// TIA Portal V17 export
// export: Created 2025-06-26T07:49:50.4539602Z, ExportSetting WithDefaults, DisplayName Totally Integrated Automation Portal, DisplayVersion V17 Update 8, DisplayName TIA Portal Openness, DisplayVersion V17 Update 8, DisplayName TIA Portal Version Control Interface, DisplayVersion V17, DisplayName STEP 7 Professional, DisplayVersion V17 Update 8, DisplayName STEP 7 Safety, DisplayVersion V17 Update 6, DisplayName WinCC Advanced, DisplayVersion V17 Update 8
DATA_BLOCK "DB_DI"   // DB2
{ S7_Optimized_Access := 'TRUE' }
AUTHOR : Heaten
VERSION : 0.1
// stored: AutoNumber true, DBAccessibleFromOPCUA true, DBAccessibleFromWebserver true, IsOnlyStoredInLoadMemory false, IsRetainMemResEnabled false, IsWriteProtectedInAS false, MemoryReserve 0
   VAR RETAIN
      SafetyRelayStatus { S7_SetPoint := 'True'} : "stDigitalInput";   // Emergency Stop status
      HBL_FS_01 { S7_SetPoint := 'True'} : "stDigitalInput";   // Flow switch heat source
      HBL_FS_02 { S7_SetPoint := 'True'} : "stDigitalInput";   // Flow switch heat sink
      HBL_EC_01_X1 { S7_SetPoint := 'True'} : "stDigitalInput";   // Oil heaters group 1 status
      HBL_EC_02_X1 { S7_SetPoint := 'True'} : "stDigitalInput";   // Oil heaters group 2 status
      DI08 { S7_SetPoint := 'True'} : "stDigitalInput";   // 24V Distribution status
      HBL_PS_500_X2 { S7_SetPoint := 'True'} : "stDigitalInput";   // Compressor discharge manifold A & B high pressure
      HBL_LS_01 { S7_SetPoint := 'True'} : "stDigitalInput";   // Drip pan sump A full
      HBL_LS_02 { S7_SetPoint := 'True'} : "stDigitalInput";   // Drip pan sump B full
      HBL_PZH_539 { S7_SetPoint := 'True'} : "stDigitalInput";   // Evaporator discharge pressure switch
      HBL_LS_632 { S7_SetPoint := 'True'} : "stDigitalInput";   // Oil separator stage 1 oil level high
      HBL_LS_633 { S7_SetPoint := 'True'} : "stDigitalInput";   // Oil separator stage 2 oil level high
      VPNUserConnected { S7_SetPoint := 'True'} : "stDigitalInput";   // VPN user logged in signal from VPN router
      CPC_LS_864 { S7_SetPoint := 'True'} : "stDigitalInput";
      HBL_LS_644 { S7_SetPoint := 'True'} : "stDigitalInput";   // Suction accumulator level switch
      HBL_LS_674 { S7_SetPoint := 'True'} : "stDigitalInput";   // Discharge accumulator level switch
      HBL_HV_640_X1 { S7_SetPoint := 'True'} : "stDigitalInput";   // Suction accumualtor drain valve open status
      HBL_HV_640_X2 { S7_SetPoint := 'True'} : "stDigitalInput";   // Suction accumualtor drain valve closed status
      HBL_HV_670_X1 { S7_SetPoint := 'True'} : "stDigitalInput";   // Discharge accumulator drain valve open status
      HBL_HV_670_X2 { S7_SetPoint := 'True'} : "stDigitalInput";   // Discharge accumulator drain valve closed status
      CPC_HV_852_X1 { S7_SetPoint := 'True'} : "stDigitalInput";   // CPC Cooler enable valve open status
      CPC_HV_852_X2 { S7_SetPoint := 'True'} : "stDigitalInput";   // CPC Cooler enable valve closed status
      HBL_HV_861_X1 { S7_SetPoint := 'True'} : "stDigitalInput";   // Compressor manifold drain valve open status
      HBL_HV_861_X2 { S7_SetPoint := 'True'} : "stDigitalInput";   // Compressor manifold drain valve closed status
   END_VAR
   VAR
      CPC_LSH_870A { S7_SetPoint := 'True'} : "stDigitalInput";   // CPC manifold refrigerant level upper
      CPC_LSL_870B { S7_SetPoint := 'True'} : "stDigitalInput";   // CPC manifold refrigernat level lower
      CPC_PZH_874 { S7_SetPoint := 'True'} : "stDigitalInput";   // CPC manifold pressure switch
   END_VAR
BEGIN
   HBL_PS_500_X2.bValueOnError := true;
END_DATA_BLOCK
